# B&R Automation Studio project Nerehta_Forming
Automation Studio 4.2.2.134; Default project

## Configuration Simulation

CPU , AutomationRuntime D4.22

### Task classes (Cpu.sw)
```
Libraries: AsIecCon, astime
```

### Hardware
```
PC_any : PC_any v1.1.0.0 (OrderNumber=PC)
  Cyclic1Duration = 100000
  Cyclic1Tolerance = 10000000
  Cyclic2Duration = 200000
  Cyclic2Tolerance = 10000000
  Cyclic3Duration = 500000
  Cyclic3Tolerance = 10000000
  Cyclic4Duration = 1000000
  Cyclic4Tolerance = 10000000
  Cyclic5Duration = 2000000
  Cyclic5Tolerance = 10000000
  Cyclic6Duration = 3000000
  Cyclic6Tolerance = 12000000
  Cyclic7Duration = 4000000
  Cyclic7Tolerance = 12000000
  Cyclic8Duration = 5000000
  Cyclic8Tolerance = 30000000
```

## Configuration X20CP1484_1

CPU X20CP1484-1, AutomationRuntime U3.09, Build 4.1.2, Vc V4.22.0

### Task classes (Cpu.sw)
```

```

### Hardware
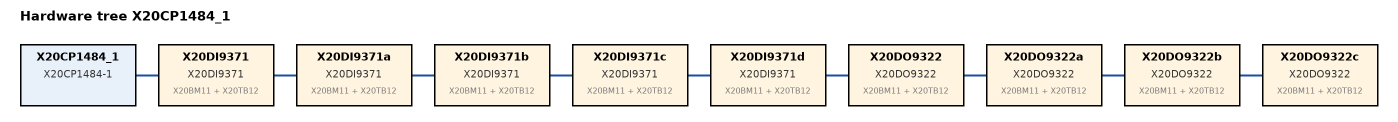
```
X20BM11 : X20BM11 v1.0.0.0  [X2X1 -> X20CP1484_1.IF6]
X20BM11a : X20BM11 v1.0.0.0  [X2X1 -> X20BM11.X2X2]
X20BM11b : X20BM11 v1.0.0.0  [X2X1 -> X20BM11a.X2X2]
X20BM11c : X20BM11 v1.0.0.0  [X2X1 -> X20BM11b.X2X2]
X20BM11d : X20BM11 v1.0.0.0  [X2X1 -> X20BM11c.X2X2]
X20BM11e : X20BM11 v1.0.0.0  [X2X1 -> X20BM11d.X2X2]
X20BM11f : X20BM11 v1.0.0.0  [X2X1 -> X20BM11e.X2X2]
X20BM11g : X20BM11 v1.0.0.0  [X2X1 -> X20BM11f.X2X2]
X20BM11h : X20BM11 v1.0.0.0  [X2X1 -> X20BM11g.X2X2]
X20CP1484_1 : X20CP1484-1 v1.1.4.0
  Cyclic1Duration = 10000
  Cyclic1Tolerance = 10000
  Cyclic2Duration = 20000
  Cyclic2Tolerance = 20000
  Cyclic3Duration = 50000
  Cyclic3Tolerance = 50000
  Cyclic4Duration = 100000
  Cyclic4Tolerance = 100000
  Cyclic5Duration = 200000
  Cyclic5Tolerance = 200000
  Cyclic6Duration = 500000
  Cyclic6Tolerance = 500000
  Cyclic7Duration = 1000000
  Cyclic7Tolerance = 1000000
  Cyclic8Duration = 10000
  Cyclic8Tolerance = 30000000
X20DI9371 : X20DI9371 v1.0.1.2  [SS1 -> X20TB12.SS; SL -> X20BM11.SL1]
X20DI9371a : X20DI9371 v1.0.1.2  [SS1 -> X20TB12a.SS; SL -> X20BM11a.SL1]
X20DI9371b : X20DI9371 v1.0.1.2  [SS1 -> X20TB12b.SS; SL -> X20BM11b.SL1]
X20DI9371c : X20DI9371 v1.0.1.2  [SS1 -> X20TB12c.SS; SL -> X20BM11c.SL1]
X20DI9371d : X20DI9371 v1.0.1.2  [SS1 -> X20TB12d.SS; SL -> X20BM11d.SL1]
X20DO9322 : X20DO9322 v1.0.2.2  [SS1 -> X20TB12e.SS; SL -> X20BM11e.SL1]
X20DO9322a : X20DO9322 v1.0.2.2  [SS1 -> X20TB12f.SS; SL -> X20BM11f.SL1]
X20DO9322b : X20DO9322 v1.0.2.2  [SS1 -> X20TB12g.SS; SL -> X20BM11g.SL1]
X20DO9322c : X20DO9322 v1.0.2.2  [SS1 -> X20TB12h.SS; SL -> X20BM11h.SL1]
X20TB12 : X20TB12 v1.0.0.0
X20TB12a : X20TB12 v1.0.0.0
X20TB12b : X20TB12 v1.0.0.0
X20TB12c : X20TB12 v1.0.0.0
X20TB12d : X20TB12 v1.0.0.0
X20TB12e : X20TB12 v1.0.0.0
X20TB12f : X20TB12 v1.0.0.0
X20TB12g : X20TB12 v1.0.0.0
X20TB12h : X20TB12 v1.0.0.0
```

## Configuration X20CP1584

CPU X20CP1584, AutomationRuntime D4.22, Build 4.1.2, Vc V4.22.0

### Task classes (Cpu.sw)
```
Cyclic#4 (cycle 100000 us, tolerance 100000 us):
  Excavator <- Excavator.prg
  Conveyor <- Conveyor.prg
  FeederBunk <- FeederBunker.prg
  Mixer <- Mixer.prg
  GrinderCla <- GrinderClay.prg
  PressScrew <- PressScrew.prg
  Control <- Control.prg
```

### Hardware
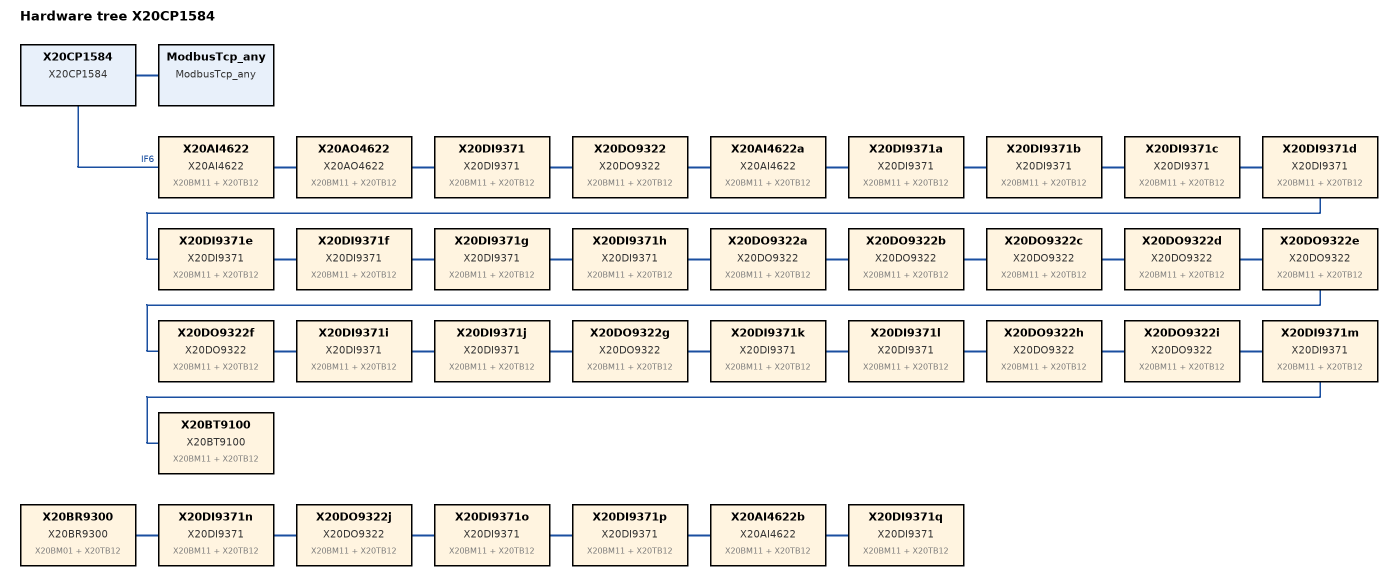
```
ModbusTcp_any : ModbusTcp_any v1.0.4.6  [ETH1 -> X20CP1584.IF2 (NodeNumber=1)]
  Cb_1
  Cb_1_FunCode = 1
X20AI4622 : X20AI4622 v1.0.2.1  [SS1 -> X20TB12.SS; SL -> X20BM11.SL1]
X20AI4622a : X20AI4622 v1.0.2.1  [SS1 -> X20TB12d.SS; SL -> X20BM11d.SL1]
X20AI4622b : X20AI4622 v1.0.2.1  [SS1 -> X20TB12ag.SS; SL -> X20BM11af.SL1]
X20AO4622 : X20AO4622 v1.0.4.1  [SS1 -> X20TB12a.SS; SL -> X20BM11a.SL1]
X20BM01 : X20BM01 v1.0.0.1
X20BM11 : X20BM11 v1.0.0.0  [X2X1 -> X20CP1584.IF6]
X20BM11a : X20BM11 v1.0.0.0  [X2X1 -> X20BM11.X2X2]
X20BM11aa : X20BM11 v1.0.0.0  [X2X1 -> X20BM11z.X2X2]
X20BM11ab : X20BM11 v1.0.0.0  [X2X1 -> X20BM01.X2X2]
X20BM11ac : X20BM11 v1.0.0.0  [X2X1 -> X20BM11ab.X2X2]
X20BM11ad : X20BM11 v1.0.0.0  [X2X1 -> X20BM11ac.X2X2]
X20BM11ae : X20BM11 v1.0.0.0  [X2X1 -> X20BM11ad.X2X2]
X20BM11af : X20BM11 v1.0.0.0  [X2X1 -> X20BM11ae.X2X2]
X20BM11ag : X20BM11 v1.0.0.0  [X2X1 -> X20BM11af.X2X2]
X20BM11b : X20BM11 v1.0.0.0  [X2X1 -> X20BM11a.X2X2]
X20BM11c : X20BM11 v1.0.0.0  [X2X1 -> X20BM11b.X2X2]
X20BM11d : X20BM11 v1.0.0.0  [X2X1 -> X20BM11c.X2X2]
X20BM11e : X20BM11 v1.0.0.0  [X2X1 -> X20BM11d.X2X2]
X20BM11f : X20BM11 v1.0.0.0  [X2X1 -> X20BM11e.X2X2]
X20BM11g : X20BM11 v1.0.0.0  [X2X1 -> X20BM11f.X2X2]
X20BM11h : X20BM11 v1.0.0.0  [X2X1 -> X20BM11g.X2X2]
X20BM11i : X20BM11 v1.0.0.0  [X2X1 -> X20BM11h.X2X2]
X20BM11j : X20BM11 v1.0.0.0  [X2X1 -> X20BM11i.X2X2]
X20BM11k : X20BM11 v1.0.0.0  [X2X1 -> X20BM11j.X2X2]
X20BM11l : X20BM11 v1.0.0.0  [X2X1 -> X20BM11k.X2X2]
X20BM11m : X20BM11 v1.0.0.0  [X2X1 -> X20BM11l.X2X2]
X20BM11n : X20BM11 v1.0.0.0  [X2X1 -> X20BM11m.X2X2]
X20BM11o : X20BM11 v1.0.0.0  [X2X1 -> X20BM11n.X2X2]
X20BM11p : X20BM11 v1.0.0.0  [X2X1 -> X20BM11o.X2X2]
X20BM11q : X20BM11 v1.0.0.0  [X2X1 -> X20BM11p.X2X2]
X20BM11r : X20BM11 v1.0.0.0  [X2X1 -> X20BM11q.X2X2]
X20BM11s : X20BM11 v1.0.0.0  [X2X1 -> X20BM11r.X2X2]
X20BM11t : X20BM11 v1.0.0.0  [X2X1 -> X20BM11s.X2X2]
X20BM11u : X20BM11 v1.0.0.0  [X2X1 -> X20BM11t.X2X2]
X20BM11v : X20BM11 v1.0.0.0  [X2X1 -> X20BM11u.X2X2]
X20BM11w : X20BM11 v1.0.0.0  [X2X1 -> X20BM11v.X2X2]
X20BM11x : X20BM11 v1.0.0.0  [X2X1 -> X20BM11w.X2X2]
X20BM11y : X20BM11 v1.0.0.0  [X2X1 -> X20BM11x.X2X2]
X20BM11z : X20BM11 v1.0.0.0  [X2X1 -> X20BM11y.X2X2]
X20BR9300 : X20BR9300 v1.0.2.6  [SS1 -> X20TB12ab.SS; SL -> X20BM01.SL1; X2X1 -> X20BT9100.X2X1]
X20BT9100 : X20BT9100 v1.0.2.3  [SS1 -> X20TB12aa.SS; SL -> X20BM11aa.SL1]
X20CP1584 : X20CP1584 v1.1.0.0
  Connector IF2:
    ActivateDevice = 1
    EthInterfaceRedundant = 0
    ActivateModbus = 1
    NumSlaves = -1
    NumAllBlocks = -1
    MemSizeIn = -1
    MemSizeOut = -1
  Connector IF3:
    EplInterfaceRedundant = 0
    EplEthInterfaceRedundant = 0
  Simulation = 1
  TimerDeviceType = SWIOTIMER
  Cyclic1Duration = 10000
  Cyclic1Tolerance = 10000
  Cyclic2Duration = 20000
  Cyclic2Tolerance = 20000
  Cyclic3Duration = 50000
  Cyclic3Tolerance = 50000
  Cyclic4Duration = 100000
  Cyclic4Tolerance = 100000
  Cyclic5Duration = 200000
  Cyclic5Tolerance = 200000
  Cyclic6Duration = 500000
  Cyclic6Tolerance = 500000
  Cyclic7Duration = 1000000
  Cyclic7Tolerance = 1000000
  Cyclic8Duration = 10000
  Cyclic8Tolerance = 30000000
X20DI9371 : X20DI9371 v1.0.1.2  [SS1 -> X20TB12b.SS; SL -> X20BM11b.SL1]
X20DI9371a : X20DI9371 v1.0.1.2  [SS1 -> X20TB12e.SS; SL -> X20BM11e.SL1]
X20DI9371b : X20DI9371 v1.0.1.2  [SS1 -> X20TB12f.SS; SL -> X20BM11f.SL1]
X20DI9371c : X20DI9371 v1.0.1.2  [SS1 -> X20TB12g.SS; SL -> X20BM11g.SL1]
X20DI9371d : X20DI9371 v1.0.1.2  [SS1 -> X20TB12h.SS; SL -> X20BM11h.SL1]
X20DI9371e : X20DI9371 v1.0.1.2  [SS1 -> X20TB12i.SS; SL -> X20BM11i.SL1]
X20DI9371f : X20DI9371 v1.0.1.2  [SS1 -> X20TB12j.SS; SL -> X20BM11j.SL1]
X20DI9371g : X20DI9371 v1.0.1.2  [SS1 -> X20TB12k.SS; SL -> X20BM11k.SL1]
X20DI9371h : X20DI9371 v1.0.1.2  [SS1 -> X20TB12l.SS; SL -> X20BM11l.SL1]
X20DI9371i : X20DI9371 v1.0.1.2  [SS1 -> X20TB12s.SS; SL -> X20BM11s.SL1]
X20DI9371j : X20DI9371 v1.0.1.2  [SS1 -> X20TB12t.SS; SL -> X20BM11t.SL1]
X20DI9371k : X20DI9371 v1.0.1.2  [SS1 -> X20TB12v.SS; SL -> X20BM11v.SL1]
X20DI9371l : X20DI9371 v1.0.1.2  [SS1 -> X20TB12w.SS; SL -> X20BM11w.SL1]
X20DI9371m : X20DI9371 v1.0.1.2  [SS1 -> X20TB12z.SS; SL -> X20BM11z.SL1]
X20DI9371n : X20DI9371 v1.0.1.2  [SS1 -> X20TB12ac.SS; SL -> X20BM11ab.SL1]
X20DI9371o : X20DI9371 v1.0.1.2  [SS1 -> X20TB12ae.SS; SL -> X20BM11ad.SL1]
X20DI9371p : X20DI9371 v1.0.1.2  [SS1 -> X20TB12af.SS; SL -> X20BM11ae.SL1]
X20DI9371q : X20DI9371 v1.0.1.2  [SS1 -> X20TB12ah.SS; SL -> X20BM11ag.SL1]
X20DO9322 : X20DO9322 v1.0.2.2  [SS1 -> X20TB12c.SS; SL -> X20BM11c.SL1]
X20DO9322a : X20DO9322 v1.0.2.2  [SS1 -> X20TB12m.SS; SL -> X20BM11m.SL1]
X20DO9322b : X20DO9322 v1.0.2.2  [SS1 -> X20TB12n.SS; SL -> X20BM11n.SL1]
X20DO9322c : X20DO9322 v1.0.2.2  [SS1 -> X20TB12o.SS; SL -> X20BM11o.SL1]
X20DO9322d : X20DO9322 v1.0.2.2  [SS1 -> X20TB12p.SS; SL -> X20BM11p.SL1]
X20DO9322e : X20DO9322 v1.0.2.2  [SS1 -> X20TB12q.SS; SL -> X20BM11q.SL1]
X20DO9322f : X20DO9322 v1.0.2.2  [SS1 -> X20TB12r.SS; SL -> X20BM11r.SL1]
X20DO9322g : X20DO9322 v1.0.2.2  [SS1 -> X20TB12u.SS; SL -> X20BM11u.SL1]
X20DO9322h : X20DO9322 v1.0.2.2  [SS1 -> X20TB12x.SS; SL -> X20BM11x.SL1]
X20DO9322i : X20DO9322 v1.0.2.2  [SS1 -> X20TB12y.SS; SL -> X20BM11y.SL1]
X20DO9322j : X20DO9322 v1.0.2.2  [SS1 -> X20TB12ad.SS; SL -> X20BM11ac.SL1]
X20TB12 : X20TB12 v1.0.0.0
X20TB12a : X20TB12 v1.0.0.0
X20TB12aa : X20TB12 v1.0.0.0
X20TB12ab : X20TB12 v1.0.0.0
X20TB12ac : X20TB12 v1.0.0.0
X20TB12ad : X20TB12 v1.0.0.0
X20TB12ae : X20TB12 v1.0.0.0
X20TB12af : X20TB12 v1.0.0.0
X20TB12ag : X20TB12 v1.0.0.0
X20TB12ah : X20TB12 v1.0.0.0
X20TB12b : X20TB12 v1.0.0.0
X20TB12c : X20TB12 v1.0.0.0
X20TB12d : X20TB12 v1.0.0.0
X20TB12e : X20TB12 v1.0.0.0
X20TB12f : X20TB12 v1.0.0.0
X20TB12g : X20TB12 v1.0.0.0
X20TB12h : X20TB12 v1.0.0.0
X20TB12i : X20TB12 v1.0.0.0
X20TB12j : X20TB12 v1.0.0.0
X20TB12k : X20TB12 v1.0.0.0
X20TB12l : X20TB12 v1.0.0.0
X20TB12m : X20TB12 v1.0.0.0
X20TB12n : X20TB12 v1.0.0.0
X20TB12o : X20TB12 v1.0.0.0
X20TB12p : X20TB12 v1.0.0.0
X20TB12q : X20TB12 v1.0.0.0
X20TB12r : X20TB12 v1.0.0.0
X20TB12s : X20TB12 v1.0.0.0
X20TB12t : X20TB12 v1.0.0.0
X20TB12u : X20TB12 v1.0.0.0
X20TB12v : X20TB12 v1.0.0.0
X20TB12w : X20TB12 v1.0.0.0
X20TB12x : X20TB12 v1.0.0.0
X20TB12y : X20TB12 v1.0.0.0
X20TB12z : X20TB12 v1.0.0.0
```

### IoMap.iom - X20CP1584/IoMap.iom
```iecst
(*********************************************************************************
 * Copyright: kiryandr
 * Author:    vzylevich
 * Created:   September 21, 2015/3:53 PM
 *********************************************************************************
 * IO mapping
 *********************************************************************************)
VAR_CONFIG
	::PressScrew:H214_Current_AI AT %IW."X20AI4622".AnalogInput01;
	::PressScrew:H214_RPM_AI AT %IW."X20AI4622".AnalogInput02;
	::PressScrew:H214_CurrentMixer_AI AT %IW."X20AI4622".AnalogInput03;
	::PressScrew:H214_RPMMixer_AI AT %IW."X20AI4622".AnalogInput04;
	::PressScrew:H214_RPM_AO AT %QW."X20AO4622".AnalogOutput01;
	::PressScrew:H214_RPMMixer_AO AT %QW."X20AO4622".AnalogOutput02;
	::GrinderCla:H211_RPM_AO AT %QW."X20AO4622".AnalogOutput03;
	::Control:H01_ControlVoltage_DI AT %IX."X20DI9371".DigitalInput01;
	::Control:H01_FuseVoltage_DI AT %IX."X20DI9371".DigitalInput02;
	::Control:H01_BAutoManMode_DI AT %IX."X20DI9371".DigitalInput03;
	::Control:H01_AutoControl_DI AT %IX."X20DI9371".DigitalInput04;
	::Control:H01_Switcher1On_DI AT %IX."X20DI9371".DigitalInput05;
	::Control:H01_BSignalLamp_DI AT %IX."X20DI9371".DigitalInput06;
	::Control:H01_BAutoStart_DI AT %IX."X20DI9371".DigitalInput09;
	::Control:H01_BAutoStop_DI AT %IX."X20DI9371".DigitalInput10;
	::Control:H01_BMoveMatStart1_DI AT %IX."X20DI9371".DigitalInput11;
	::Control:H01_BMoveMatStop1_DI AT %IX."X20DI9371".DigitalInput12;
	::Control:H01_PrDeviceVolt_DO AT %QX."X20DO9322".DigitalOutput01;
	::Control:H01_LampVoltage_DO AT %QX."X20DO9322".DigitalOutput02;
	::Control:H01_LampPreAutoMan_DO AT %QX."X20DO9322".DigitalOutput03;
	::Control:H01_LampAutoModeOn_DO AT %QX."X20DO9322".DigitalOutput04;
	::Control:H01_PreAutoOn_DO AT %QX."X20DO9322".DigitalOutput05;
	::Control:H01_Reset_DO AT %QX."X20DO9322".DigitalOutput06;
	::Control:H01_LampFault_DO AT %QX."X20DO9322".DigitalOutput07;
	::Control:H01_SoundForming_DO AT %QX."X20DO9322".DigitalOutput08;
	::Control:H01_LampAutoMode_DO AT %QX."X20DO9322".DigitalOutput09;
	::Control:H01_LampMoveMat1On_DO AT %QX."X20DO9322".DigitalOutput10;
	::Control:H01_LampMoveMat1Mode_DO AT %QX."X20DO9322".DigitalOutput11;
	::Control:H01_LampExplEnd_DO AT %QX."X20DO9322".DigitalOutput12;
	::GrinderCla:H211_Current_AI AT %IW."X20AI4622a".AnalogInput01;
	::GrinderCla:H211_RPM_AI AT %IW."X20AI4622a".AnalogInput02;
	::Control:H01_BFailure_DI AT %IX."X20DI9371a".DigitalInput01;
	::Control:H01_BExplEnd_DI AT %IX."X20DI9371a".DigitalInput02;
	::Control:H01_BMoveMatStart2_DI AT %IX."X20DI9371a".DigitalInput03;
	::Control:H01_BMoveMatStop2_DI AT %IX."X20DI9371a".DigitalInput04;
	::Control:H01_PrMagnV_DI AT %IX."X20DI9371a".DigitalInput06;
	::Control:H01_PneumSw_DI AT %IX."X20DI9371a".DigitalInput07;
	::Control:H01_ZeroP_DI AT %IX."X20DI9371a".DigitalInput08;
	::Control:H01_ZeroP2_DI AT %IX."X20DI9371a".DigitalInput09;
	::Control:H01_ZeroPRustik_DI AT %IX."X20DI9371a".DigitalInput10;
	::Excavator:H201_zeroP_DI AT %IX."X20DI9371a".DigitalInput11;
	::Excavator:H201_fault_DI AT %IX."X20DI9371a".DigitalInput12;
	::Control:H01_PrElmVacP_DI AT %IX."X20DI9371b".DigitalInput02;
	::PressScrew:H214_TurnBPumpVacOn_DI AT %IX."X20DI9371b".DigitalInput03;
	::PressScrew:H214_TurnBPumpVacOff_DI AT %IX."X20DI9371b".DigitalInput04;
	::Control:H01_Winding_DI AT %IX."X20DI9371b".DigitalInput05;
	::Control:H01_TempVacP_DI AT %IX."X20DI9371b".DigitalInput06;
	::Control:H01_Filter_DI AT %IX."X20DI9371b".DigitalInput07;
	::Control:H01_WLevelMax_DI AT %IX."X20DI9371b".DigitalInput08;
	::Control:H01_WLevelMin_DI AT %IX."X20DI9371b".DigitalInput09;
	::PressScrew:H214_PrElmMove_DI AT %IX."X20DI9371c".DigitalInput01;
	::PressScrew:H214_SwLampUp_DI AT %IX."X20DI9371c".DigitalInput02;
	::PressScrew:H214_SwLampDown_DI AT %IX."X20DI9371c".DigitalInput03;
	::PressScrew:H214_TopSw_DI AT %IX."X20DI9371c".DigitalInput04;
	::PressScrew:H214_BottomSw_DI AT %IX."X20DI9371c".DigitalInput05;
	::PressScrew:H214_PrElmMixer_DI AT %IX."X20DI9371c".DigitalInput07;
	::PressScrew:H214_TurnBMixerOn_DI AT %IX."X20DI9371c".DigitalInput09;
	::PressScrew:H214_TurnBElmOff2_DI AT %IX."X20DI9371c".DigitalInput10;
	::PressScrew:H214_ThyristorMixer_DI AT %IX."X20DI9371c".DigitalInput11;
	::PressScrew:H214_ThyristorSomething_DI AT %IX."X20DI9371c".DigitalInput12;
	::PressScrew:H214_SwLampMixer_DI AT %IX."X20DI9371d".DigitalInput01;
	::PressScrew:H214_SlipClutch_DI AT %IX."X20DI9371d".DigitalInput02;
	::PressScrew:H214_IrrigMixer_DI AT %IX."X20DI9371d".DigitalInput03;
	::Conveyor:H212_PrElmOn_DI AT %IX."X20DI9371d".DigitalInput04;
	::Conveyor:H212_ElmBeltStart_DI AT %IX."X20DI9371d".DigitalInput05;
	::Conveyor:H209_ElmStartStop_DI AT %IX."X20DI9371d".DigitalInput06;
	::Conveyor:H212_Ready_DI AT %IX."X20DI9371d".DigitalInput07;
	::Conveyor:H212_DownControl_DI AT %IX."X20DI9371d".DigitalInput08;
	::GrinderCla:H211_PrElmOn_DI AT %IX."X20DI9371d".DigitalInput09;
	::GrinderCla:H211_TurnBOn_DI AT %IX."X20DI9371d".DigitalInput10;
	::GrinderCla:H211_TurnBOff_DI AT %IX."X20DI9371d".DigitalInput11;
	::GrinderCla:H211_ThyristorW_DI AT %IX."X20DI9371d".DigitalInput12;
	::GrinderCla:H211_Thyristor_DI AT %IX."X20DI9371e".DigitalInput01;
	::GrinderCla:H211_PrOilpElmOn_DI AT %IX."X20DI9371e".DigitalInput02;
	::GrinderCla:H211_PressureOilp_DI AT %IX."X20DI9371e".DigitalInput03;
	::GrinderCla:H211_PrTarelElmOn_DI AT %IX."X20DI9371e".DigitalInput04;
	::GrinderCla:H211_LightDevice_DI AT %IX."X20DI9371e".DigitalInput05;
	::GrinderCla:H211_LightSwithcer_DI AT %IX."X20DI9371e".DigitalInput06;
	::GrinderCla:H211_MetalCover_DI AT %IX."X20DI9371e".DigitalInput07;
	::GrinderCla:H211_SlipControl_DI AT %IX."X20DI9371e".DigitalInput08;
	::GrinderCla:H211_MaterialControl_DI AT %IX."X20DI9371e".DigitalInput09;
	::GrinderCla:H211_Irrig_DI AT %IX."X20DI9371e".DigitalInput10;
	::GrinderCla:H211_Max_DI AT %IX."X20DI9371e".DigitalInput11;
	::GrinderCla:H211_Min_DI AT %IX."X20DI9371e".DigitalInput12;
	::Conveyor:H212_PrElmBottom_DI AT %IX."X20DI9371f".DigitalInput01;
	::Conveyor:H212_LightForward_DI AT %IX."X20DI9371f".DigitalInput02;
	::Conveyor:H212_LightBackward_DI AT %IX."X20DI9371f".DigitalInput03;
	::Conveyor:H212_BordersControl_DI AT %IX."X20DI9371f".DigitalInput04;
	::Conveyor:H212_MoveControl_DI AT %IX."X20DI9371f".DigitalInput05;
	::Conveyor:H212_MetDetector_DI AT %IX."X20DI9371f".DigitalInput06;
	::Conveyor:H217_LightBottom_DI AT %IX."X20DI9371f".DigitalInput08;
	::Conveyor:H217_PrElm_DI AT %IX."X20DI9371g".DigitalInput01;
	::Conveyor:H217_Light_DI AT %IX."X20DI9371g".DigitalInput02;
	::Conveyor:H217_PrElmOn_DI AT %IX."X20DI9371g".DigitalInput08;
	::Conveyor:H215_Light_DI AT %IX."X20DI9371g".DigitalInput07;
	::Control:H02_Control_DI AT %IX."X20DI9371g".DigitalInput06;
	::Control:H02_SS1_DI AT %IX."X20DI9371g".DigitalInput05;
	::Conveyor:H217_Ready_DI AT %IX."X20DI9371g".DigitalInput09;
	::Conveyor:H216_Light_DI AT %IX."X20DI9371g".DigitalInput10;
	::Conveyor:H217_DownControl_DI AT %IX."X20DI9371g".DigitalInput11;
	::Conveyor:H217_BordersControl_DI AT %IX."X20DI9371g".DigitalInput12;
	::PressScrew:H214_ElmOilpOn_DI AT %IX."X20DI9371h".DigitalInput02;
	::Conveyor:H217_Start_DI AT %IX."X20DI9371h".DigitalInput03;
	::Control:H01_Bypass1_DI AT %IX."X20DI9371h".DigitalInput04;
	::Control:H01_Bypass2_DI AT %IX."X20DI9371h".DigitalInput05;
	::Control:H01_Ident1_DI AT %IX."X20DI9371h".DigitalInput06;
	::Control:H01_Ident2_DI AT %IX."X20DI9371h".DigitalInput07;
	::Control:H01_Ident3_DI AT %IX."X20DI9371h".DigitalInput08;
	::Control:H01_ElmWPumpOn_DI AT %IX."X20DI9371h".DigitalInput09;
	::GrinderCla:H211_PressureOilpOn_DI AT %IX."X20DI9371h".DigitalInput10;
	::GrinderCla:H211_TarelElmOn_DI AT %IX."X20DI9371h".DigitalInput11;
	::Control:H01_LampMoveMat2On_DO AT %QX."X20DO9322a".DigitalOutput01;
	::Control:H01_LampMoveMat2Mode_DO AT %QX."X20DO9322a".DigitalOutput02;
	::PressScrew:H214_WetSideOn_DO AT %QX."X20DO9322a".DigitalOutput03;
	::Excavator:H201_Remote_DO AT %QX."X20DO9322a".DigitalOutput04;
	::PressScrew:H214_Rustik1_DO AT %QX."X20DO9322a".DigitalOutput05;
	::PressScrew:H214_Rustik2_DO AT %QX."X20DO9322a".DigitalOutput06;
	::Control:H01_Bypass1_DO AT %QX."X20DO9322a".DigitalOutput07;
	::Control:H01_Bypass2_DO AT %QX."X20DO9322a".DigitalOutput08;
	::PressScrew:H214_StartStop_DO AT %QX."X20DO9322a".DigitalOutput09;
	::Mixer:H208_MixerStartStop_DO AT %QX."X20DO9322a".DigitalOutput10;
	::Control:H01_LampWetSide_DO AT %QX."X20DO9322a".DigitalOutput11;
	::Excavator:H201_Lamp_DO AT %QX."X20DO9322a".DigitalOutput12;
	::PressScrew:H214_ElmVacP_DO AT %QX."X20DO9322b".DigitalOutput01;
	::PressScrew:H214_LampVacP_DO AT %QX."X20DO9322b".DigitalOutput02;
	::PressScrew:H214_MValveW_DO AT %QX."X20DO9322b".DigitalOutput03;
	::PressScrew:H214_ElmWPump_DO AT %QX."X20DO9322b".DigitalOutput04;
	::PressScrew:H214_ThyristorControl_DO AT %QX."X20DO9322b".DigitalOutput05;
	::PressScrew:H214_LampElm_DO AT %QX."X20DO9322b".DigitalOutput06;
	::PressScrew:H214_ElmTransmCoil_DO AT %QX."X20DO9322b".DigitalOutput07;
	::PressScrew:H214_LampPressureOil_DO AT %QX."X20DO9322b".DigitalOutput08;
	::PressScrew:H214_ElmOilp_DO AT %QX."X20DO9322b".DigitalOutput09;
	::PressScrew:H214_LampOilp_DO AT %QX."X20DO9322b".DigitalOutput10;
	::PressScrew:H214_PressureV_DO AT %QX."X20DO9322b".DigitalOutput11;
	::PressScrew:H214_PressureW_DO AT %QX."X20DO9322b".DigitalOutput12;
	::PressScrew:H214_LampClutch_DO AT %QX."X20DO9322c".DigitalOutput01;
	::PressScrew:H214_ElmSpeedUp_DO AT %QX."X20DO9322c".DigitalOutput02;
	::PressScrew:H214_LampSpeedUp_DO AT %QX."X20DO9322c".DigitalOutput03;
	::PressScrew:H214_ElmSpeedDown_DO AT %QX."X20DO9322c".DigitalOutput04;
	::PressScrew:H214_LampSpeedDown_DO AT %QX."X20DO9322c".DigitalOutput05;
	::PressScrew:H214_ThyristorMixer_DO AT %QX."X20DO9322c".DigitalOutput06;
	::PressScrew:H214_LampMixer_DO AT %QX."X20DO9322c".DigitalOutput07;
	::PressScrew:H214_PressureVMixer_DO AT %QX."X20DO9322c".DigitalOutput08;
	::PressScrew:H214_PressureVWMixer_DO AT %QX."X20DO9322c".DigitalOutput09;
	::PressScrew:H214_LampMixerClutch_DO AT %QX."X20DO9322c".DigitalOutput10;
	::PressScrew:H214_IrrigV_DO AT %QX."X20DO9322c".DigitalOutput11;
	::PressScrew:H214_LampIrrigMixer_DO AT %QX."X20DO9322c".DigitalOutput12;
	::Conveyor:H212_Forward_DO AT %QX."X20DO9322d".DigitalOutput01;
	::Conveyor:H212_LampForward_DO AT %QX."X20DO9322d".DigitalOutput02;
	::Conveyor:H212_Backward_DO AT %QX."X20DO9322d".DigitalOutput03;
	::Conveyor:H212_LampBackward_DO AT %QX."X20DO9322d".DigitalOutput04;
	::GrinderCla:H211_ThyristorControl_DO AT %QX."X20DO9322d".DigitalOutput05;
	::GrinderCla:H211_ElmLamp_DO AT %QX."X20DO9322d".DigitalOutput06;
	::GrinderCla:H211_OilpStartStop_DO AT %QX."X20DO9322d".DigitalOutput07;
	::GrinderCla:H211_OilpLamp_DO AT %QX."X20DO9322d".DigitalOutput08;
	::GrinderCla:H211_ClaygrinderStartStop_DO AT %QX."X20DO9322d".DigitalOutput09;
	::GrinderCla:H211_ClaygrinderLamp_DO AT %QX."X20DO9322d".DigitalOutput10;
	::GrinderCla:H211_ClutchVPressure_DO AT %QX."X20DO9322d".DigitalOutput11;
	::GrinderCla:H211_ClutchLamp_DO AT %QX."X20DO9322e".DigitalOutput01;
	::GrinderCla:H211_ClutchW_DO AT %QX."X20DO9322e".DigitalOutput02;
	::GrinderCla:H211_BeltDW_DO AT %QX."X20DO9322e".DigitalOutput03;
	::GrinderCla:H211_IrrigV_DO AT %QX."X20DO9322e".DigitalOutput04;
	::GrinderCla:H211_IrrigLamp_DO AT %QX."X20DO9322e".DigitalOutput05;
	::GrinderCla:H211_Irrig_DO AT %QX."X20DO9322e".DigitalOutput06;
	::GrinderCla:H211_Irrig_DO AT %QX."X20DO9322e".DigitalOutput07;
	::Control:H03_PreStart1_DO AT %QX."X20DO9322e".DigitalOutput08;
	::Control:H03_LampPreStart1_DO AT %QX."X20DO9322e".DigitalOutput09;
	::Control:H03_PreStart2_DO AT %QX."X20DO9322e".DigitalOutput10;
	::Control:H03_LampPreStart2_DO AT %QX."X20DO9322e".DigitalOutput11;
	::GrinderCla:H211_StartStop_DO AT %QX."X20DO9322e".DigitalOutput12;
	::Control:H01_SocketOn_DO AT %QX."X20DO9322f".DigitalOutput01;
	::Conveyor:H217_StartStop_DO AT %QX."X20DO9322f".DigitalOutput03;
	::Conveyor:H202_Lamp_DO AT %QX."X20DO9322f".DigitalOutput04;
	::Conveyor:H212_LampBelt2_DO AT %QX."X20DO9322f".DigitalOutput05;
	::Conveyor:H215_Lamp_DO AT %QX."X20DO9322f".DigitalOutput06;
	::Conveyor:H216_Lamp_DO AT %QX."X20DO9322f".DigitalOutput08;
	::Conveyor:H213_PrElmOn_DI AT %IX."X20DI9371i".DigitalInput06;
	::Conveyor:H213_Ready_DI AT %IX."X20DI9371i".DigitalInput07;
	::Conveyor:H213_DownControl_DI AT %IX."X20DI9371i".DigitalInput08;
	::Conveyor:H213_BordersControl_DI AT %IX."X20DI9371i".DigitalInput09;
	::Conveyor:H213_MoveControl_DI AT %IX."X20DI9371i".DigitalInput10;
	::Conveyor:H215_PrElmOn_DI AT %IX."X20DI9371j".DigitalInput01;
	::Conveyor:H215_Ready_DI AT %IX."X20DI9371j".DigitalInput02;
	::Conveyor:H215_DownControl_DI AT %IX."X20DI9371j".DigitalInput03;
	::Conveyor:H215_BordersControl_DI AT %IX."X20DI9371j".DigitalInput04;
	::Conveyor:H215_MoveControl_DI AT %IX."X20DI9371j".DigitalInput05;
	::Conveyor:H216_PrElmOn_DI AT %IX."X20DI9371j".DigitalInput06;
	::Conveyor:H216_Ready_DI AT %IX."X20DI9371j".DigitalInput07;
	::Conveyor:H216_DownControl_DI AT %IX."X20DI9371j".DigitalInput08;
	::Conveyor:H216_BordersControl_DI AT %IX."X20DI9371j".DigitalInput09;
	::Conveyor:H216_MoveControl_DI AT %IX."X20DI9371j".DigitalInput10;
	::Conveyor:H213_ElmStartStop_DO AT %QX."X20DO9322g".DigitalOutput02;
	::Conveyor:H215_ElmStartStop_DO AT %QX."X20DO9322g".DigitalOutput03;
	::Conveyor:H216_ElmStartStop_DO AT %QX."X20DO9322g".DigitalOutput04;
	::Control:H02_ManMode_DO AT %QX."X20DO9322g".DigitalOutput05;
	::Control:H02_AutoMode_DO AT %QX."X20DO9322g".DigitalOutput06;
	::Control:H02_Control_DO AT %QX."X20DO9322g".DigitalOutput07;
	::Control:H02_Fault_DO AT %QX."X20DO9322g".DigitalOutput08;
	::Control:H02_ControlCircuit_DO AT %QX."X20DO9322g".DigitalOutput09;
	::Control:H02_Permission1_DO AT %QX."X20DO9322g".DigitalOutput11;
	::Control:H02_Permission2_DO AT %QX."X20DO9322g".DigitalOutput12;
	::Control:H02_Reset_DI AT %IX."X20DI9371k".DigitalInput01;
	::Control:H02_Permission1_DI AT %IX."X20DI9371k".DigitalInput02;
	::Control:H02_Permission2_DI AT %IX."X20DI9371k".DigitalInput03;
	::Conveyor:H202_ElmBeltStart_DI AT %IX."X20DI9371k".DigitalInput04;
	::Conveyor:H203_ElmBeltStart_DI AT %IX."X20DI9371k".DigitalInput05;
	::Conveyor:H204_ElmBeltStart_DI AT %IX."X20DI9371k".DigitalInput06;
	::Conveyor:H205_ElmTranspStart_DI AT %IX."X20DI9371k".DigitalInput07;
	::Conveyor:H205_StartForwardMan_DI AT %IX."X20DI9371k".DigitalInput08;
	::Conveyor:H205_StartBackwardMan_DI AT %IX."X20DI9371k".DigitalInput09;
	::Conveyor:H207_ElmBeltStart_DI AT %IX."X20DI9371k".DigitalInput10;
	::Mixer:H208_ElmStart_DI AT %IX."X20DI9371l".DigitalInput01;
	::Mixer:H208_ElmStop_DI AT %IX."X20DI9371l".DigitalInput02;
	::Mixer:H208_ClutchOn_DI AT %IX."X20DI9371l".DigitalInput03;
	::Mixer:H208_ValveWOn_DI AT %IX."X20DI9371l".DigitalInput04;
	::Mixer:H208_OilpStart_DI AT %IX."X20DI9371l".DigitalInput05;
	::Mixer:H208_OilpStop_DI AT %IX."X20DI9371l".DigitalInput06;
	::Conveyor:H202_Ready_DO AT %QX."X20DO9322h".DigitalOutput01;
	::Conveyor:H202_ElmOn_DO AT %QX."X20DO9322h".DigitalOutput02;
	::Conveyor:H203_Ready_DO AT %QX."X20DO9322h".DigitalOutput03;
	::Conveyor:H203_ElmOn_DO AT %QX."X20DO9322h".DigitalOutput04;
	::Conveyor:H204_Ready_DO AT %QX."X20DO9322h".DigitalOutput05;
	::Conveyor:H204_ElmOn_DO AT %QX."X20DO9322h".DigitalOutput06;
	::Conveyor:H205_Ready_DO AT %QX."X20DO9322h".DigitalOutput07;
	::Conveyor:H205_TranspElmOn_DO AT %QX."X20DO9322h".DigitalOutput08;
	::Conveyor:H205_CombElmForwOn_DO AT %QX."X20DO9322h".DigitalOutput09;
	::Conveyor:H205_CombElmBackwOn_DO AT %QX."X20DO9322h".DigitalOutput10;
	::Conveyor:H207_Ready_DO AT %QX."X20DO9322h".DigitalOutput11;
	::Conveyor:H207_ElmOn_DO AT %QX."X20DO9322h".DigitalOutput12;
	::Mixer:H208_Ready_DO AT %QX."X20DO9322i".DigitalOutput01;
	::Mixer:H208_ElmOn_DO AT %QX."X20DO9322i".DigitalOutput02;
	::Mixer:H208_Overload_DO AT %QX."X20DO9322i".DigitalOutput03;
	::Mixer:H208_OilPressureNorm_DO AT %QX."X20DO9322i".DigitalOutput04;
	::Mixer:H208_Normal_DO AT %QX."X20DO9322i".DigitalOutput05;
	::Mixer:H208_ClutchOnInd_DO AT %QX."X20DO9322i".DigitalOutput06;
	::Mixer:H208_ValveWOnInd_DO AT %QX."X20DO9322i".DigitalOutput07;
	::PressScrew:H214_PrElmOn_DI AT %IX."X20DI9371m".DigitalInput01;
	::PressScrew:H214_TurnBOn_DI AT %IX."X20DI9371m".DigitalInput02;
	::PressScrew:H214_TurnBElmOff_DI AT %IX."X20DI9371m".DigitalInput03;
	::PressScrew:H214_ThyristorMode_DI AT %IX."X20DI9371m".DigitalInput04;
	::PressScrew:H214_ThyristorCooler_DI AT %IX."X20DI9371m".DigitalInput05;
	::PressScrew:H214_PrElmChassis_DI AT %IX."X20DI9371m".DigitalInput06;
	::PressScrew:H214_PressureOilp_DI AT %IX."X20DI9371m".DigitalInput07;
	::PressScrew:H214_PrElmOilp_DI AT %IX."X20DI9371m".DigitalInput08;
	::PressScrew:H214_PressureOilp2_DI AT %IX."X20DI9371m".DigitalInput09;
	::PressScrew:H214_SwLampClutch_DI AT %IX."X20DI9371m".DigitalInput10;
	::PressScrew:H214_SlipControl_DI AT %IX."X20DI9371m".DigitalInput11;
	::PressScrew:H214_HighMax_DI AT %IX."X20DI9371m".DigitalInput12;
	::Conveyor:H203_PrElmOn_DI AT %IX."X20DI9371n".DigitalInput01;
	::Conveyor:H203_Ready_DI AT %IX."X20DI9371n".DigitalInput02;
	::Conveyor:H203_DownControl_DI AT %IX."X20DI9371n".DigitalInput03;
	::Conveyor:H203_BordersControl_DI AT %IX."X20DI9371n".DigitalInput04;
	::Conveyor:H203_MoveControl_DI AT %IX."X20DI9371n".DigitalInput05;
	::Conveyor:H204_PrElmOn_DI AT %IX."X20DI9371n".DigitalInput06;
	::Conveyor:H204_Ready_DI AT %IX."X20DI9371n".DigitalInput07;
	::Conveyor:H204_DownControl_DI AT %IX."X20DI9371n".DigitalInput08;
	::Conveyor:H204_BordersControl_DI AT %IX."X20DI9371n".DigitalInput09;
	::Conveyor:H204_MoveControl_DI AT %IX."X20DI9371n".DigitalInput10;
	::Conveyor:H203_ElmStartStop_DO AT %QX."X20DO9322j".DigitalOutput01;
	::Conveyor:H204_ElmStartStop_DO AT %QX."X20DO9322j".DigitalOutput02;
	::Conveyor:H205_ElmStartStop_DO AT %QX."X20DO9322j".DigitalOutput03;
	::Conveyor:H205_StartForward_DO AT %QX."X20DO9322j".DigitalOutput04;
	::Conveyor:H205_StartBackward_DO AT %QX."X20DO9322j".DigitalOutput05;
	::Mixer:H208_ElmStartStop_DO AT %QX."X20DO9322j".DigitalOutput06;
	::Mixer:H208_OilpStartStop_DO AT %QX."X20DO9322j".DigitalOutput07;
	::Mixer:H208_ClutchOn_DO AT %QX."X20DO9322j".DigitalOutput08;
	::Mixer:H208_ValveWOn_DO AT %QX."X20DO9322j".DigitalOutput09;
	::Conveyor:H202_ElmStartStop_DO AT %QX."X20DO9322j".DigitalOutput10;
	::Conveyor:H209_ElmStartStop_DO AT %QX."X20DO9322j".DigitalOutput11;
	::Conveyor:H207_ElmStartStop_DO AT %QX."X20DO9322j".DigitalOutput12;
	::Conveyor:H205_PrElmOn_DI AT %IX."X20DI9371o".DigitalInput01;
	::Conveyor:H205_TransporterOn_DI AT %IX."X20DI9371o".DigitalInput02;
	::Conveyor:H205_StartForward_DI AT %IX."X20DI9371o".DigitalInput03;
	::Conveyor:H205_StartBackward_DI AT %IX."X20DI9371o".DigitalInput04;
	::Conveyor:H205_Ready_DI AT %IX."X20DI9371o".DigitalInput05;
	::Conveyor:H205_CombControl_DI AT %IX."X20DI9371o".DigitalInput06;
	::Conveyor:H202_PrElmOn_DI AT %IX."X20DI9371o".DigitalInput07;
	::Conveyor:H202_Ready_DI AT %IX."X20DI9371o".DigitalInput08;
	::Conveyor:H202_DownControl_DI AT %IX."X20DI9371o".DigitalInput09;
	::Conveyor:H202_BordersControl_DI AT %IX."X20DI9371o".DigitalInput10;
	::Conveyor:H202_MoveControl_DI AT %IX."X20DI9371o".DigitalInput11;
	::Conveyor:H202_MaterialControl_DI AT %IX."X20DI9371o".DigitalInput12;
	::Mixer:H208_PressureNon_DI AT %IX."X20DI9371p".DigitalInput01;
	::Mixer:H208_PrOn_DI AT %IX."X20DI9371p".DigitalInput03;
	::Mixer:H208_ElmOn_DI AT %IX."X20DI9371p".DigitalInput04;
	::Mixer:H208_ProElmOilpOn_DI AT %IX."X20DI9371p".DigitalInput05;
	::Mixer:H208_OilpOn_DI AT %IX."X20DI9371p".DigitalInput06;
	::Conveyor:H209_PrElmOn_DI AT %IX."X20DI9371p".DigitalInput07;
	::Conveyor:H209_Ready_DI AT %IX."X20DI9371p".DigitalInput08;
	::Conveyor:H209_DownControl_DI AT %IX."X20DI9371p".DigitalInput09;
	::Conveyor:H209_BordersControl_DI AT %IX."X20DI9371p".DigitalInput10;
	::Conveyor:H209_MoveControl_DI AT %IX."X20DI9371p".DigitalInput11;
	::Mixer:H208_CurrentBControl_AI AT %IW."X20AI4622b".AnalogInput02;
	::Conveyor:H207_PrElmOn_DI AT %IX."X20DI9371q".DigitalInput01;
	::Conveyor:H207_Ready_DI AT %IX."X20DI9371q".DigitalInput02;
	::Conveyor:H207_DownControl_DI AT %IX."X20DI9371q".DigitalInput03;
	::Conveyor:H207_BordersControl_DI AT %IX."X20DI9371q".DigitalInput04;
	::Conveyor:H207_MoveControl_DI AT %IX."X20DI9371q".DigitalInput05;
END_VAR
```

## Logical view

Binary libraries used (declarations not repeated): RUNTIME, OPERATOR, AsIecCon, astime


### Program Logical/Excavator (ANSIC)

#### Cyclic.c - Cyclic code
```c
#include <bur/plctypes.h>

#ifdef _DEFAULT_INCLUDES
	#include <AsDefault.h>
#endif

void _CYCLIC ProgramCyclic(void)
{

}
```

#### Init.c - Initialization code
```c
#include <bur/plctypes.h>

#ifdef _DEFAULT_INCLUDES
	#include <AsDefault.h>
#endif

void _INIT ProgramInit(void)
{

}
```

#### Exit.c - Exit code
```c
#include <bur/plctypes.h>

#ifdef _DEFAULT_INCLUDES
	#include <AsDefault.h>
#endif

void _EXIT ProgramExit(void)
{

}
```

#### Variables.var - Local variables
```iecst
VAR
	H201_Lamp_DO : BOOL := FALSE;
	H201_zeroP_DI : BOOL := FALSE;
	H201_fault_DI : BOOL := FALSE;
	H201_Remote_DO : BOOL := FALSE;
	H201_protectUp_DI : BOOL := FALSE;
	H201_pressureUp_DI : BOOL := FALSE;
	H201_Up_DI : BOOL := FALSE;
	H201_Down_DI : BOOL := FALSE;
	H201_BoxOff_DI : BOOL := FALSE;
	H201_mechUp_DI : BOOL := FALSE;
	H201_upMechOut_DI : BOOL := FALSE;
	H201_upMechDown_DI : BOOL := FALSE;
	H201_endLeft_DI : BOOL := FALSE;
	H201_endRight_DI : BOOL := FALSE;
	H201_wallLeft_DI : BOOL := FALSE;
	H201_QSlLeft_DI : BOOL := FALSE;
	H201_wallRight_DI : BOOL := FALSE;
	H201_QSlRight_DI : BOOL := FALSE;
	H201_prElmotor1_DI : BOOL := FALSE;
	H201_prElmotor2_DI : BOOL := FALSE;
	H201_faultInvertor_DI : BOOL := FALSE;
	H201_prPullElm_DI : BOOL := FALSE;
	H201_pullElmSlLeft_DI : BOOL := FALSE;
	H201_pullElmSlRight_DI : BOOL := FALSE;
	H201_pullElmSlFrom_DI : BOOL := FALSE;
	H201_pullElmQLeft_DI : BOOL := FALSE;
	H201_pullElmQRight_DI : BOOL := FALSE;
	H201_pullElmQFrom_DI : BOOL := FALSE;
	H201_prElmCounterAP_DI : BOOL := FALSE;
	H201_counterAPElm1_DI : BOOL := FALSE;
	H201_counterAPElm2_DI : BOOL := FALSE;
	H201_OverloadElm1_DI : BOOL := FALSE;
	H201_OverloadElm2_DI : BOOL := FALSE;
	H201_MValveLeft_DI : BOOL := FALSE;
	H201_MValveRight_DI : BOOL := FALSE;
	H201_PrElmUnit_DI : BOOL := FALSE;
	H201_LubrChain_DI : BOOL := FALSE;
	H201_MonitorHigh_DI : BOOL := FALSE;
	H201_PressureOil_DI : BOOL := FALSE;
	H201_DetectB1_DI : BOOL := FALSE;
	H201_DetectB2_DI : BOOL := FALSE;
	H201_DetectB3_DI : BOOL := FALSE;
	H201_DetectB4_DI : BOOL := FALSE;
	H201_ControlVolt_DO : BOOL := FALSE;
	H201_ControlVoltW_DO : BOOL := FALSE;
	H201_PreManMode_DO : BOOL := FALSE;
	H201_PreAutoMode_DO : BOOL := FALSE;
	H201_PreRemoteMode_DO : BOOL := FALSE;
	H201_AutoStart_DO : BOOL := FALSE;
	H201_Siren_DO : BOOL := FALSE;
	H201_FlashLight_DO : BOOL := FALSE;
	H201_AutoMode_DO : BOOL := FALSE;
	H201_WFPressureOil_DO : BOOL := FALSE;
	H201_WFCircuit_DO : BOOL := FALSE;
	H201_FSecCircuit_DO : BOOL := FALSE;
	H201_FLoad_DO : BOOL := FALSE;
	H201_Elm1p2_DO : BOOL := FALSE;
	H201_FDiagnostic_DO : BOOL := FALSE;
	H201_ChainUp_DO : BOOL := FALSE;
	H201_WFChainUp_DO : BOOL := FALSE;
	H201_ChainDown_DO : BOOL := FALSE;
	H201_WFChainDown_DO : BOOL := FALSE;
	H201_BucketUp_DO : BOOL := FALSE;
	H201_BucketDown_DO : BOOL := FALSE;
	H201_LeftBorder_DO : BOOL := FALSE;
	H201_RightBorder_DO : BOOL := FALSE;
	H201_MBoxLeft_DO : BOOL := FALSE;
	H201_MBoxRight_DO : BOOL := FALSE;
	H201_BorderSl_DO : BOOL := FALSE;
	H201_BorderF_DO : BOOL := FALSE;
	H201_BorderTRight_DO : BOOL := FALSE;
	H201_BorderTLeft_DO : BOOL := FALSE;
	H201_LabrUnit_DO : BOOL := FALSE;
	H201_OilLevel_DO : BOOL := FALSE;
	H201_LubrChain_DO : BOOL := FALSE;
	H201_ExcBox1_DO : BOOL := FALSE;
	H201_ExcBox2_DO : BOOL := FALSE;
	H201_ExcBox3_DO : BOOL := FALSE;
	H201_UnlockVIn_DI : BOOL := FALSE;
	H201_UnlockV_DI : BOOL := FALSE;
	H201_ManPreStart_DI : BOOL := FALSE;
	H201_AutoPreStart_DI : BOOL := FALSE;
	H201_RemotePreStart_DI : BOOL := FALSE;
	H201_SoundIn_DI : BOOL := FALSE;
	H201_SoundOut_DI : BOOL := FALSE;
	H201_Reset_DI : BOOL := FALSE;
	H201_AutoStart_DI : BOOL := FALSE;
	H201_AutoStop_DI : BOOL := FALSE;
	H201_RemoteResol_DI : BOOL := FALSE;
	H201_PrCircuit1_DI : BOOL := FALSE;
	H201_SecCircuit_DI : BOOL := FALSE;
	H201_ExplCircuit_DI : BOOL := FALSE;
	H201_LampTest_DI : BOOL := FALSE;
	H201_CircuitIn_DI : BOOL := FALSE;
	H201_CircuitOut_DI : BOOL := FALSE;
	H201_ChainDown_DI : BOOL := FALSE;
END_VAR
```

### Program Logical/Conveyor (ANSIC)

#### lib.h
```c
/*
	Проверка блокировок:
  	если сработала одна из блокировок возвращает 1, иначе 0
*/
BOOL blockingCheck(BOOL PrElmOn, BOOL DownControl, BOOL BordersControl, BOOL MoveControl)
{
	BOOL out;
	out = 0;
	if (PrElmOn || DownControl || BordersControl || MoveControl)
		out = 1;

	return out;
}

/*
	Запуск конвейера
	ConvStart - переменная DO, которая запускает данный конвейер
*/
void convH2XXStart(BOOL ConvStart)
{
	ConvStart = 1;
}

/*
	Остановка конвейера
	ConvStart - переменная DO, которая запускает данный конвейер
*/
void convH2XXStop(BOOL ConvStart)
{
	ConvStart = 0;
}

/*
	convH2XX_DO_B - переменная привязываемая к кнопке панели, отвечающая за запуск конвейера ("Пуск/Стоп")
*/
void convH2XX(BOOL PrElmOn, BOOL DownControl, BOOL BordersControl, BOOL MoveControl, BOOL Mode, BOOL Ready, BOOL ElmBeltStart,
	BOOL ConvStart)
{
	if (!blockingCheck(PrElmOn, DownControl, BordersControl, MoveControl) &&
		convH2XX_DO_B)
		convH2XXStart(ConvStart);
	else convH2XXStop(ConvStart);
}
```

#### Cyclic.c - Cyclic code
```c
#include <bur/plctypes.h>
#include <lib.h>

#ifdef _DEFAULT_INCLUDES
	#include <AsDefault.h>
#endif

void _CYCLIC ProgramCyclic(void)
{
	/*Блок обработки работы конвейера H202*/
	void convH202()
	{

	}
	/*Блок обработки работы конвейера H203*/
	void convH203()
	{

	}
	/*Блок обработки работы конвейера H204*/
	void convH204()
	{

	}
	/*Блок обработки работы конвейера H207*/
	void convH207()
	{

	}
	/*Блок обработки работы конвейера H209*/
	void convH209()
	{

	}
	/*Блок обработки работы конвейера H212*/
	void convH212()
	{

	}
	/*Блок обработки работы конвейера H213*/
	void convH213()
	{

	}
	/*Блок обработки работы конвейера H215*/
	void convH215()
	{

	}
	/*Блок обработки работы конвейера H216*/
	void convH216()
	{

	}
	/*Блок обработки работы конвейера H217*/
	void convH217()
	{

	}
}
```

#### Init.c - Initialization code
```c
#include <bur/plctypes.h>

#ifdef _DEFAULT_INCLUDES
	#include <AsDefault.h>
#endif

void _INIT ProgramInit(void)
{

}
```

#### Exit.c - Exit code
```c
#include <bur/plctypes.h>

#ifdef _DEFAULT_INCLUDES
	#include <AsDefault.h>
#endif

void _EXIT ProgramExit(void)
{

}
```

#### Variables.var - Local variables
```iecst
(*Conv 202*)
VAR
	H202_Light_DI : BOOL := FALSE;
	H202_Lamp_DO : BOOL := FALSE;
	H202_PrElmOn_DI : BOOL := FALSE;
	H202_ElmStartStop_DO : BOOL := FALSE;
	H202_Ready_DI : BOOL := FALSE;
	H202_DownControl_DI : BOOL := FALSE;
	H202_BordersControl_DI : BOOL := FALSE;
	H202_MoveControl_DI : BOOL := FALSE;
	H202_MaterialControl_DI : BOOL := FALSE;
	H202_ElmBeltStart_DI : BOOL := FALSE;
	H202_Ready_DO : BOOL := FALSE;
	H202_ElmOn_DO : BOOL := FALSE;
	H202_Start_DI : BOOL := FALSE;
END_VAR
(*Conv 203*)
VAR
	H203_ElmOn_DO : BOOL := FALSE;
	H203_PrElmOn_DI : BOOL := FALSE;
	H203_ElmStartStop_DO : BOOL := FALSE;
	H203_Ready_DI : BOOL := FALSE;
	H203_DownControl_DI : BOOL := FALSE;
	H203_BordersControl_DI : BOOL := FALSE;
	H203_MoveControl_DI : BOOL := FALSE;
	H203_ElmBeltStart_DI : BOOL := FALSE;
	H203_Ready_DO : BOOL := FALSE;
END_VAR
(*Conv 204*)
VAR
	H204_ElmOn_DO : BOOL := FALSE;
	H204_PrElmOn_DI : BOOL := FALSE;
	H204_ElmStartStop_DO : BOOL := FALSE;
	H204_Ready_DI : BOOL := FALSE;
	H204_DownControl_DI : BOOL := FALSE;
	H204_BordersControl_DI : BOOL := FALSE;
	H204_MoveControl_DI : BOOL := FALSE;
	H204_ElmBeltStart_DI : BOOL := FALSE;
	H204_Ready_DO : BOOL := FALSE;
END_VAR
(*Conv 205*)
VAR
	H205_ElmStartStop_DO : BOOL := FALSE;
	H205_StartForward_DO : BOOL := FALSE;
	H205_StartBackward_DO : BOOL := FALSE;
	H205_PrElmOn_DI : BOOL := FALSE;
	H205_TransporterOn_DI : BOOL := FALSE;
	H205_StartForward_DI : BOOL := FALSE;
	H205_StartBackward_DI : BOOL := FALSE;
	H205_Ready_DI : BOOL := FALSE;
	H205_CombControl_DI : BOOL := FALSE;
	H205_ElmTranspStart_DI : BOOL := FALSE;
	H205_StartForwardMan_DI : BOOL := FALSE;
	H205_StartBackwardMan_DI : BOOL := FALSE;
	H205_Ready_DO : BOOL := FALSE;
	H205_TranspElmOn_DO : BOOL := FALSE;
	H205_CombElmBackwOn_DO : BOOL := FALSE;
	H205_CombElmForwOn_DO : BOOL := FALSE;
END_VAR
(*Conv 207*)
VAR
	H207_PrElmOn_DI : BOOL := FALSE;
	H207_ElmStartStop_DO : BOOL := FALSE;
	H207_Ready_DI : BOOL := FALSE;
	H207_DownControl_DI : BOOL := FALSE;
	H207_BordersControl_DI : BOOL := FALSE;
	H207_MoveControl_DI : BOOL := FALSE;
	H207_ElmBeltStart_DI : BOOL := FALSE;
	H207_Ready_DO : BOOL := FALSE;
	H207_ElmOn_DO : BOOL := FALSE;
END_VAR
(*Conv 209*)
VAR
	H209_ElmStartStop_DI : BOOL := FALSE;
	H209_PrElmOn_DI : BOOL := FALSE;
	H209_ElmStartStop_DO : BOOL := FALSE;
	H209_Ready_DI : BOOL := FALSE;
	H209_DownControl_DI : BOOL := FALSE;
	H209_BordersControl_DI : BOOL := FALSE;
	H209_MoveControl_DI : BOOL := FALSE;
END_VAR
(*Conv 212*)
VAR
	H212_ElmBeltStart_DI : BOOL := FALSE;
	H212_LightForward_DI : BOOL := FALSE;
	H212_Ready_DI : BOOL := FALSE;
	H212_DownControl_DI : BOOL := FALSE;
	H212_BordersControl_DI : BOOL := FALSE;
	H212_MoveControl_DI : BOOL := FALSE;
	H212_LightBackward_DI : BOOL := FALSE;
	H212_LampForward_DO : BOOL := FALSE;
	H212_LampBackward_DO : BOOL := FALSE;
	H212_LampBelt2_DO : BOOL := FALSE;
	H212_PrElmOn_DI : BOOL := FALSE;
	H212_Forward_DO : BOOL := FALSE;
	H212_Backward_DO : BOOL := FALSE;
	H212_PrElmBottom_DI : BOOL := FALSE;
	H212_MetDetector_DI : BOOL := FALSE;
END_VAR
(*Conv 213*)
VAR
	H213_PrElmOn_DI : BOOL := FALSE;
	H213_ElmStartStop_DO : BOOL := FALSE;
	H213_Ready_DI : BOOL := FALSE;
	H213_DownControl_DI : BOOL := FALSE;
	H213_BordersControl_DI : BOOL := FALSE;
	H213_MoveControl_DI : BOOL := FALSE;
END_VAR
(*Conv 215*)
VAR
	H215_PrElmOn_DI : BOOL := FALSE;
	H215_ElmStartStop_DO : BOOL := FALSE;
	H215_Ready_DI : BOOL := FALSE;
	H215_DownControl_DI : BOOL := FALSE;
	H215_BordersControl_DI : BOOL := FALSE;
	H215_MoveControl_DI : BOOL := FALSE;
	H215_Light_DI : BOOL := FALSE;
	H215_Lamp_DO : BOOL := FALSE;
END_VAR
(*Conv 216*)
VAR
	H216_PrElmOn_DI : BOOL := FALSE;
	H216_ElmStartStop_DO : BOOL := FALSE;
	H216_Ready_DI : BOOL := FALSE;
	H216_DownControl_DI : BOOL := FALSE;
	H216_BordersControl_DI : BOOL := FALSE;
	H216_MoveControl_DI : BOOL := FALSE;
	H216_Light_DI : BOOL := FALSE;
	H216_Lamp_DO : BOOL := FALSE;
END_VAR
(*Conv 217*)
VAR
	H217_PrElm_DI : BOOL := FALSE;
	H217_PrElmOn_DI : BOOL := FALSE;
	H217_ElmStartStop_DO : BOOL := FALSE;
	H217_Ready_DI : BOOL := FALSE;
	H217_DownControl_DI : BOOL := FALSE;
	H217_BordersControl_DI : BOOL := FALSE;
	H217_MoveControl_DI : BOOL := FALSE;
	H217_LightBottom_DI : BOOL := FALSE;
	H217_Light_DI : BOOL := FALSE;
	H217_Start_DI : BOOL := FALSE;
	H217_StartStop_DO : BOOL := FALSE;
	New_Variable49 : BOOL := FALSE;
	New_Variable50 : BOOL := FALSE;
	New_Variable51 : BOOL := FALSE;
	New_Variable52 : BOOL := FALSE;
	New_Variable : BOOL := FALSE;
END_VAR
```

### Program Logical/FeederBunker (ANSIC)

#### Cyclic.c - Cyclic code
```c
#include <bur/plctypes.h>

#ifdef _DEFAULT_INCLUDES
	#include <AsDefault.h>
#endif

void _CYCLIC ProgramCyclic(void)
{

}
```

#### Init.c - Initialization code
```c
#include <bur/plctypes.h>

#ifdef _DEFAULT_INCLUDES
	#include <AsDefault.h>
#endif

void _INIT ProgramInit(void)
{

}
```

#### Exit.c - Exit code
```c
#include <bur/plctypes.h>

#ifdef _DEFAULT_INCLUDES
	#include <AsDefault.h>
#endif

void _EXIT ProgramExit(void)
{

}
```

#### Variables.var - Local variables
```iecst
VAR
	H205_ElmStartStop_DO : BOOL := FALSE;
	H205_StartForward_DO : BOOL := FALSE;
	H205_StartBackward_DO : BOOL := FALSE;
	H205_PrElmOn_DI : BOOL := FALSE;
	H205_TransporterOn_DI : BOOL := FALSE;
	H205_StartForward_DI : BOOL := FALSE;
	H205_StartBackward_DI : BOOL := FALSE;
	H205_Ready_DI : BOOL := FALSE;
	H205_CombControl_DI : BOOL := FALSE;
	H205_ElmTranspStart_DI : BOOL := FALSE;
	H205_StartForwardMan_DI : BOOL := FALSE;
	H205_StartBackwardMan_DI : BOOL := FALSE;
	H205_Ready_DO : BOOL := FALSE;
	H205_TranspElmOn_DO : BOOL := FALSE;
	H205_CombElmBackwOn_DO : BOOL := FALSE;
	H205_CombElmForwOn_DO : BOOL := FALSE;
END_VAR
```

### Program Logical/Mixer (ANSIC)

#### Cyclic.c - Cyclic code
```c
#include <bur/plctypes.h>

#ifdef _DEFAULT_INCLUDES
	#include <AsDefault.h>
#endif

void _CYCLIC ProgramCyclic(void)
{

}
```

#### Init.c - Initialization code
```c
#include <bur/plctypes.h>

#ifdef _DEFAULT_INCLUDES
	#include <AsDefault.h>
#endif

void _INIT ProgramInit(void)
{

}
```

#### Exit.c - Exit code
```c
#include <bur/plctypes.h>

#ifdef _DEFAULT_INCLUDES
	#include <AsDefault.h>
#endif

void _EXIT ProgramExit(void)
{

}
```

#### Variables.var - Local variables
```iecst
VAR
	H208_ClutchOn_DO : BOOL := FALSE;
	H208_ElmStartStop_DO : BOOL := FALSE;
	H208_OilpStartStop_DO : BOOL := FALSE;
	H208_ClutchStarting_DO : BOOL := FALSE;
	H208_ValveWOn_DO : BOOL := FALSE;
	H208_CurrentBControl_AI : INT := 0;
	H208_PrOn_DI : BOOL := FALSE;
	H208_ElmOn_DI : BOOL := FALSE;
	H208_ProElmOilpOn_DI : BOOL := FALSE;
	H208_OilpOn_DI : BOOL := FALSE;
	H208_PressureNon_DI : BOOL := FALSE;
	H208_ElmStart_DI : BOOL := FALSE;
	H208_ElmStop_DI : BOOL := FALSE;
	H208_ClutchOn_DI : BOOL := FALSE;
	H208_ValveWOn_DI : BOOL := FALSE;
	H208_OilpStart_DI : BOOL := FALSE;
	H208_OilpStop_DI : BOOL := FALSE;
	H208_Ready_DO : BOOL := FALSE;
	H208_ElmOn_DO : BOOL := FALSE;
	H208_Overload_DO : BOOL := FALSE;
	H208_OilPressureNorm_DO : BOOL := FALSE;
	H208_Normal_DO : BOOL := FALSE;
	H208_ClutchOnInd_DO : BOOL := FALSE;
	H208_ValveWOnInd_DO : BOOL := FALSE;
	H208_MixerStartStop_DO : BOOL := FALSE;
END_VAR
```

### Program Logical/GrinderClay (ANSIC)

#### Cyclic.c - Cyclic code
```c
#include <bur/plctypes.h>

#ifdef _DEFAULT_INCLUDES
	#include <AsDefault.h>
#endif

void _CYCLIC ProgramCyclic(void)
{

}
```

#### Init.c - Initialization code
```c
#include <bur/plctypes.h>

#ifdef _DEFAULT_INCLUDES
	#include <AsDefault.h>
#endif

void _INIT ProgramInit(void)
{

}
```

#### Exit.c - Exit code
```c
#include <bur/plctypes.h>

#ifdef _DEFAULT_INCLUDES
	#include <AsDefault.h>
#endif

void _EXIT ProgramExit(void)
{

}
```

#### Variables.var - Local variables
```iecst
VAR
	H211_Current_AI : INT := 0;
	H211_RPM_AI : INT := 0;
	H211_RPM_AO : INT := 0;
	H211_Irrig_DI : BOOL := FALSE;
	H211_TurnBOn_DI : BOOL := FALSE;
	H211_TurnBOff_DI : BOOL := FALSE;
	H211_LightDevice_DI : BOOL := FALSE;
	H211_LightSwithcer_DI : BOOL := FALSE;
	H211_Irrig_DO : BOOL := FALSE;
	H211_IrrigLamp_DO : BOOL := FALSE;
	H211_ElmLamp_DO : BOOL := FALSE;
	H211_OilpLamp_DO : BOOL := FALSE;
	H211_ClaygrinderLamp_DO : BOOL := FALSE;
	H211_ClutchLamp_DO : BOOL := FALSE;
	H211_PrElmOn_DI : BOOL := FALSE;
	H211_ThyristorW_DI : BOOL := FALSE;
	H211_Thyristor_DI : BOOL := FALSE;
	H211_PrOilpElmOn_DI : BOOL := FALSE;
	H211_PressureOilp_DI : BOOL := FALSE;
	H211_PrTarelElmOn_DI : BOOL := FALSE;
	H211_SlipControl_DI : BOOL := FALSE;
	H211_MaterialControl_DI : BOOL := FALSE;
	H211_Max_DI : BOOL := FALSE;
	H211_Min_DI : BOOL := FALSE;
	H211_PressureOilpOn_DI : BOOL := FALSE;
	H211_TarelElmOn_DI : BOOL := FALSE;
	H211_ThyristorControl_DO : BOOL := FALSE;
	H211_OilpStartStop_DO : BOOL := FALSE;
	H211_ClaygrinderStartStop_DO : BOOL := FALSE;
	H211_ClutchVPressure_DO : BOOL := FALSE;
	H211_ClutchVPressureW_DO : BOOL := FALSE;
	H211_ClutchW_DO : BOOL := FALSE;
	H211_BeltDW_DO : BOOL := FALSE;
	H211_IrrigV_DO : BOOL := FALSE;
	H211_StartStop_DO : BOOL := FALSE;
	H211_MetalCover_DI : BOOL := FALSE;
END_VAR
```

### Program Logical/PressScrew (ANSIC)

#### Cyclic.c - Cyclic code
```c
#include <bur/plctypes.h>

#ifdef _DEFAULT_INCLUDES
	#include <AsDefault.h>
#endif

void _CYCLIC ProgramCyclic(void)
{

}
```

#### Init.c - Initialization code
```c
#include <bur/plctypes.h>

#ifdef _DEFAULT_INCLUDES
	#include <AsDefault.h>
#endif

void _INIT ProgramInit(void)
{

}
```

#### Exit.c - Exit code
```c
#include <bur/plctypes.h>

#ifdef _DEFAULT_INCLUDES
	#include <AsDefault.h>
#endif

void _EXIT ProgramExit(void)
{

}
```

#### Variables.var - Local variables
```iecst
VAR
	H214_Current_AI : INT := 0;
	H214_RPM_AI : INT := 0;
	H214_RPM_AO : INT := 0;
	H214_CurrentMixer_AI : INT := 0;
	H214_RPMMixer_AI : INT := 0;
	H214_RPMMixer_AO : INT := 0;
	H214_TurnBElmOff2_DI : BOOL := FALSE;
	H214_SwLampClutch_DI : BOOL := FALSE;
	H214_SwLampDown_DI : BOOL := FALSE;
	H214_TurnBPumpVacOn_DI : BOOL := FALSE;
	H214_TurnBPumpVacOff_DI : BOOL := FALSE;
	H214_TurnBElmOn_DI : BOOL := FALSE;
	H214_TurnBElmOff_DI : BOOL := FALSE;
	H214_SwLampUp_DI : BOOL := FALSE;
	H214_TurnBMixerOn_DI : BOOL := FALSE;
	H214_SwLampMixer_DI : BOOL := FALSE;
	H214_LampPumpVac_DO : BOOL := FALSE;
	H214_LampPressureOil_DO : BOOL := FALSE;
	H214_LampElm_DO : BOOL := FALSE;
	H214_LampOilp_DO : BOOL := FALSE;
	H214_LampClutch_DO : BOOL := FALSE;
	H214_LampSpeedUp_DO : BOOL := FALSE;
	H214_LampSpeedDown_DO : BOOL := FALSE;
	H214_LampMixer_DO : BOOL := FALSE;
	H214_LampMixerClutch_DO : BOOL := FALSE;
	H214_PrElmOn_DI : BOOL := FALSE;
	H214_TurnBOn_DI : BOOL := FALSE;
	H214_ThyristorMode_DI : BOOL := FALSE;
	H214_ThyristorCooler_DI : BOOL := FALSE;
	H214_PrElmChassis_DI : BOOL := FALSE;
	H214_PressureOilp_DI : BOOL := FALSE;
	H214_PrElmOilp_DI : BOOL := FALSE;
	H214_PressureOilp2_DI : BOOL := FALSE;
	H214_SlipControl_DI : BOOL := FALSE;
	H214_HighMax_DI : BOOL := FALSE;
	H214_PrElmMove_DI : BOOL := FALSE;
	H214_TopSw_DI : BOOL := FALSE;
	H214_BottomSw_DI : BOOL := FALSE;
	H214_PrElmMixer_DI : BOOL := FALSE;
	H214_ThyristorMixer_DI : BOOL := FALSE;
	H214_ThyristorSomething_DI : BOOL := FALSE;
	H214_WetSideOn_DO : BOOL := FALSE;
	H214_StartStop_DO : BOOL := FALSE;
	H214_ThyristorControl_DO : BOOL := FALSE;
	H214_ElmTransmCoil_DO : BOOL := FALSE;
	H214_ElmOilp_DO : BOOL := FALSE;
	H214_PressureV_DO : BOOL := FALSE;
	H214_PressureW_DO : BOOL := FALSE;
	H214_ElmSpeedUp_DO : BOOL := FALSE;
	H214_ElmSpeedDown_DO : BOOL := FALSE;
	H214_ThyristorMixer_DO : BOOL := FALSE;
	H214_PressureVMixer_DO : BOOL := FALSE;
	H214_PressureVWMixer_DO : BOOL := FALSE;
	H214_IrrigV_DO : BOOL := FALSE;
	H214_LampIrrigMixer_DO : BOOL := FALSE;
	H214_SlipClutch_DI : BOOL := FALSE;
	H214_IrrigMixer_DI : BOOL := FALSE;
	H214_ElmOilpOn_DI : BOOL := FALSE;
	H214_Rustik1_DO : BOOL := FALSE;
	H214_Rustik2_DO : BOOL := FALSE;
	H214_ElmVacP_DO : BOOL := FALSE;
	H214_LampVacP_DO : BOOL := FALSE;
	H214_MValveW_DO : BOOL := FALSE;
	H214_ElmWPump_DO : BOOL := FALSE;
END_VAR
```

### Program Logical/Control (ANSIC)

#### Cyclic.c - Cyclic code
```c
#include <bur/plctypes.h>

#ifdef _DEFAULT_INCLUDES
	#include <AsDefault.h>
#endif

void _CYCLIC ProgramCyclic(void)
{

}
```

#### Init.c - Initialization code
```c
#include <bur/plctypes.h>

#ifdef _DEFAULT_INCLUDES
	#include <AsDefault.h>
#endif

void _INIT ProgramInit(void)
{

}
```

#### Exit.c - Exit code
```c
#include <bur/plctypes.h>

#ifdef _DEFAULT_INCLUDES
	#include <AsDefault.h>
#endif

void _EXIT ProgramExit(void)
{

}
```

#### Variables.var - Local variables
```iecst
(*Управляющие сигналы H01*)
VAR
	H01_ControlVoltage_DI : BOOL := FALSE;
	H01_AutoControl_DI : BOOL := FALSE;
	H01_BAutoStop_DI : BOOL := FALSE;
	H01_BMoveMatStop1_DI : BOOL := FALSE;
	H01_BAutoManMode_DI : BOOL := FALSE;
	H01_BAutoStart_DI : BOOL := FALSE;
	H01_BMoveMatStart1_DI : BOOL := FALSE;
	H01_BExplEnd_DI : BOOL := FALSE;
	H01_BMoveMatStart2_DI : BOOL := FALSE;
	H01_BMoveMatStop2_DI : BOOL := FALSE;
	H01_Bypass1_DI : BOOL := FALSE;
	H01_Bypass2_DI : BOOL := FALSE;
	H01_Ident1_DI : BOOL := FALSE;
	H01_Ident2_DI : BOOL := FALSE;
	H01_Ident3_DI : BOOL := FALSE;
	H01_ElmWPumpOn_DI : BOOL := FALSE;
	H01_LampMoveMat2On_DO : BOOL := FALSE;
	H01_LampWetSide_DO : BOOL := FALSE;
	H01_LampMoveMat2Mode_DO : BOOL := FALSE;
	H01_Bypass1_DO : BOOL := FALSE;
	H01_Bypass2_DO : BOOL := FALSE;
	H01_SocketOn_DO : BOOL := FALSE;
	H01_FuseVoltage_DI : BOOL := FALSE;
	H01_Switcher1On_DI : BOOL := FALSE;
	H01_BSignalLamp_DI : BOOL := FALSE;
	H01_LampVoltage_DO : BOOL := FALSE;
	H01_LampAutoMode_DO : BOOL := FALSE;
	H01_LampMoveMat1Mode_DO : BOOL := FALSE;
	H01_LampAutoModeOn_DO : BOOL := FALSE;
	H01_LampMoveMat1On_DO : BOOL := FALSE;
	H01_LampExplEnd_DO : BOOL := FALSE;
	H01_PrDeviceVolt_DO : BOOL := FALSE;
	H01_LampPreAutoMan_DO : BOOL := FALSE;
	H01_PreAutoOn_DO : BOOL := FALSE;
	H01_Reset_DO : BOOL := FALSE;
	H01_LampFault_DO : BOOL := FALSE;
	H01_SoundForming_DO : BOOL := FALSE;
	H01_BFailure_DI : BOOL := FALSE;
	H01_PrMagnV_DI : BOOL := FALSE;
	H01_PneumSw_DI : BOOL := FALSE;
	H01_ZeroP_DI : BOOL := FALSE;
	H01_ZeroP2_DI : BOOL := FALSE;
	H01_ZeroPRustik_DI : BOOL := FALSE;
	H01_PrElmVacP_DI : BOOL := FALSE;
	H01_Winding_DI : BOOL := FALSE;
	H01_TempVacP_DI : BOOL := FALSE;
	H01_Filter_DI : BOOL := FALSE;
	H01_WLevelMax_DI : BOOL := FALSE;
	H01_WLevelMin_DI : BOOL := FALSE;
END_VAR
(*Контроль состояния цепей управления H02*)
VAR
	H02_SS1_DI : BOOL := FALSE;
	H02_Control_DI : BOOL := FALSE;
	H02_ManMode_DO : BOOL := FALSE;
	H02_AutoMode_DO : BOOL := FALSE;
	H02_Control_DO : BOOL := FALSE;
	H02_Fault_DO : BOOL := FALSE;
	H02_ControlCircuit_DO : BOOL := FALSE;
	H02_Permission1_DO : BOOL := FALSE;
	H02_Permission2_DO : BOOL := FALSE;
	H02_Reset_DI : BOOL := FALSE;
	H02_Permission1_DI : BOOL := FALSE;
	H02_Permission2_DI : BOOL := FALSE;
END_VAR
(*Включение предпусковой сигнализации H03*)
VAR
	H03_PreStart1_DO : BOOL := FALSE;
	H03_PreStart2_DO : BOOL := FALSE;
	H03_LampPreStart1_DO : BOOL := FALSE;
	H03_LampPreStart2_DO : BOOL := FALSE;
END_VAR
```
